// TIA Portal project "Prueba_08-05-23_Adrian" (V16)

(* hardware
DEVICE "S7-1200 station_1"  S7-1200 Station
   slot 0: "Rack_0"  S7-1200 Rack  Rack  V1.0
   slot 1: "PLC_1"  CPU 1214C AC/DC/Rly  6ES7 214-1BE30-0XB0  V2.2
*)

// ===== PLC "PLC_1"  CPU 1214C AC/DC/Rly =====

VAR_GLOBAL   // PLC tag table "Tabla de variables estándar"
   "ENCENDIDO" AT %I0.0 : Bool;
   "CAMBIO" AT %I0.1 : Bool;
   "PARADA" AT %I0.2 : Bool;
   "KM1" AT %Q0.0 : Bool;
   "KM2" AT %Q0.1 : Bool;
   "KM3" AT %Q0.2 : Bool;
   "TERMICO" AT %I0.3 : Bool;
END_VAR

ORGANIZATION_BLOCK "Main"   // OB1, LAD, ProgramCycle
TITLE = "Main Program Sweep (Cycle)"
{ S7_Optimized_Access := 'TRUE' }
VERSION : 0.1
   VAR_TEMP   // added for the SCL form of the ladder/FBD networks
      _w1 : Bool;
   END_VAR
BEGIN

REGION Network 1
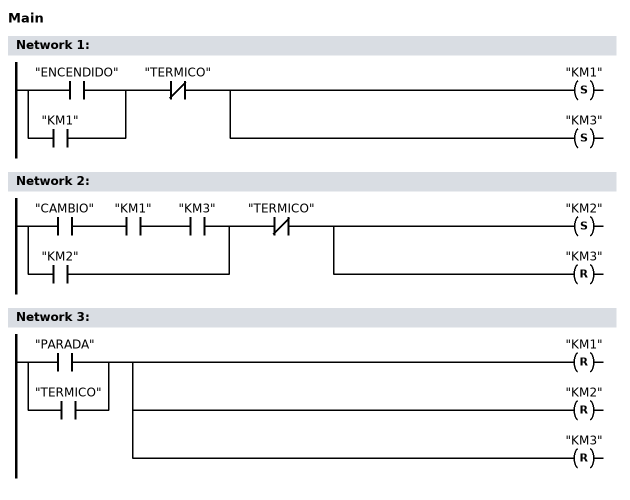
   RUNG wire#powerrail
      Contact( "ENCENDIDO" )
      wire#w1
      I_Contact( "TERMICO" )
      wire#w2
      S_Coil( "KM1" )
   END_RUNG
   RUNG wire#powerrail
      Contact( "KM1" )
   END_RUNG wire#w1
   RUNG wire#w2
      S_Coil( "KM3" )
   END_RUNG
   // the same network as SCL:
   #_w1 := ("ENCENDIDO" OR "KM1") AND NOT "TERMICO";
   IF #_w1 THEN
       "KM1" := TRUE;
       "KM3" := TRUE;
   END_IF;
END_REGION

REGION Network 2
   RUNG wire#powerrail
      Contact( "CAMBIO" )
      Contact( "KM1" )
      Contact( "KM3" )
      wire#w1
      I_Contact( "TERMICO" )
      wire#w2
      S_Coil( "KM2" )
   END_RUNG
   RUNG wire#powerrail
      Contact( "KM2" )
   END_RUNG wire#w1
   RUNG wire#w2
      R_Coil( "KM3" )
   END_RUNG
   // the same network as SCL:
   #_w1 := (("CAMBIO" AND "KM1" AND "KM3") OR "KM2") AND NOT "TERMICO";
   IF #_w1 THEN
       "KM2" := TRUE;
       "KM3" := FALSE;
   END_IF;
END_REGION

REGION Network 3
   RUNG wire#powerrail
      Contact( "PARADA" )
      wire#w1
      R_Coil( "KM1" )
   END_RUNG
   RUNG wire#powerrail
      Contact( "TERMICO" )
   END_RUNG wire#w1
   RUNG wire#w1
      R_Coil( "KM2" )
   END_RUNG
   RUNG wire#w1
      R_Coil( "KM3" )
   END_RUNG
   // the same network as SCL:
   IF "PARADA" OR "TERMICO" THEN
       "KM1" := FALSE;
       "KM2" := FALSE;
       "KM3" := FALSE;
   END_IF;
END_REGION
END_ORGANIZATION_BLOCK